FUNCTION_BLOCK AlbertsDataManager EXTENDS TcoData.TcoDataExchange
VAR
	//this variable has to called "_data" - PC app will access this variable by its name.
	_data : AlbertsSettings;
END_VAR

SUPER^();

END_FUNCTION_BLOCK

(* stored: Version 1.1.0.1, ProductVersion 3.1.4024.5
   POU AlbertsDataManager: Id {d8171ebe-c997-0d84-32d9-c05aeaa63c40}, SpecialFunc None *)
